// TwinCAT 3 PLC project VFD
// ProgramVersion: 3.1.4024.0
// libraries:
//   Modbus RTU Base, * (NewEngineer)
//   Tc2_ModbusRTU, * (Beckhoff Automation GmbH)
//   Tc2_Standard, * (Beckhoff Automation GmbH)
//   Tc2_System, * (Beckhoff Automation GmbH)
//   Tc3_Module, * (Beckhoff Automation GmbH)
//   TC3_Utilities_C, * (NewEngineer)
// project tree:
//   DUTs/ServoIpro/ E_IProCtrlMode.TcDUT (not stored), E_IProCurrentMode.TcDUT, E_IProStatus.TcDUT, E_IPro_PositionCmdModeSelection.TcDUT (not stored), E_IPro_State.TcDUT
//   DUTs/VFD/ E_VfdMdriverFaultInfor.TcDUT (not stored), E_VFD_State.TcDUT (not stored), E_VFD_Status.TcDUT (not stored)
//   / PlcTask.TcTTO
//   POUs/ FB_IPRO_ModbusRTU.TcPOU, FB_UniversalVFDModbus.TcPOU, FB_VFD_ABB_ACS480.TcPOU, FB_VFD_Mdriver.TcPOU, FB_VFD_V20_Siemens.TcPOU, I_Ipro_MotorPower.TcIO, I_UniversalVFD.TcIO, MAIN.TcPOU
//   TEST/ FB_ModbusMaster_Test.TcPOU (not stored), FB_ModbusSlave_Test.TcPOU (not stored), FB_UniversalVFDModbus_Ex.TcPOU (not stored), FB_UniversalVFDModbus_Test.TcPOU (not stored), PGR_Test.TcPOU (not stored)
// real-time tasks:
//   TASK PlcTask: cycle T#10ms, priority 20, ADS port 350

CONFIGURATION VFD
    RESOURCE PLC ON TwinCAT3
        TASK PlcTask(INTERVAL := T#10ms, PRIORITY := 20);
        PROGRAM MAIN WITH PlcTask : MAIN;
    END_RESOURCE
END_CONFIGURATION

// ---- DUTs/ServoIpro/E_IProCurrentMode.TcDUT
//{attribute 'strict'}
TYPE E_IProCurrentMode :
(
	IPRO_CURRENT_MODE_NOT_RESPONDE := -10,
	IPRO_CURRENT_MODE_POSITION		:= 0,
	IPRO_CURRENT_MODE_SPEED			:= 1,
	IPRO_CURRENT_MODE_TORQUE		:= 2
)INT := IPRO_CURRENT_MODE_NOT_RESPONDE;
END_TYPE

// ---- DUTs/ServoIpro/E_IProStatus.TcDUT
//{attribute 'strict'}
{attribute 'to_string'}
TYPE E_IProStatus :
(
	IPRO_STATUS_NOT_RESPOND := -10,
	IPRO_STATUS_INTITIZATION := 0,
	IPRO_STATUS_THE_HIGH_VOLTAGE := 1,
	IPRO_STATUS_READY			:= 2,
	IPRO_STATUS_RUN				:= 3, // OPERATION
	IPRO_STATUS_FORCED_TO_STOP	:= 4,
	IPRO_STATUS_FAULT			:= 5,
	IPRO_STATUS_STO_IN			:= 6
)INT := IPRO_STATUS_NOT_RESPOND;
END_TYPE

// ---- DUTs/ServoIpro/E_IPro_State.TcDUT
{attribute 'strict'}
{attribute 'to_string'}
TYPE E_IPro_State :
(
	IPRO_UNINITIALIZED		:= 0,	(* Axis is not prepared to work - power is off *)
	IPRO_INITIALIZING		:= 10,	(* Axis is preparing to power - reset FB and power on *)
	IPRO_READY_INITIALIZED		:= 20,	(*  *)
	IPRO_IDLE				:= 25,// MOVE DONE TO HERE
	IPRO_HOME			:= 30,	(* Axis is homing to reference point *)
	IPRO_HOME_DONE			:= 40,	(* Axis homing procedure has finished - fererence position has been found *)
	IPRO_MOVE_ABSOLUTE		:= 50,	(* Axis is moving to absolute position - discrete motion *)
	IPRO_MOVE_ABSOLUTE_DONE		:= 60,	(* Axis movement to absolute position finished *)
	IPRO_MOVE_TORQUE	:= 70,
	IPRO_MOVE_TORQUE_DONE	:= 80,
	//IPRO_MOVE_VELOCITY		:= 90,
	//IPRO_MOVE_VELOCITY_DONE	:= 100
	IPRO_STOP			:= 90,	(* Axis is stopping *)
	IPRO_STOP_DONE			:= 100,	(* Axis stopped *)
	IPRO_RESET			:= 110,	(* Axis is resseting all function blocks and occured errors *)
	IPRO_RESET_DONE			:= 120,	(* Axis reset procedure done *)
	IPRO_ABORTING			:= -10	(* Aborting *)
);
END_TYPE

// ---- POUs/I_Ipro_MotorPower.TcIO
INTERFACE I_Ipro_MotorPower

PROPERTY Active : bool
GET
END_GET
END_PROPERTY

PROPERTY Busy : bool
GET
END_GET
END_PROPERTY

PROPERTY ControlMode : E_IProCtrlMode
GET
END_GET
SET
END_SET
END_PROPERTY

PROPERTY ControlModeSwitchCmd : bool
GET
END_GET
END_PROPERTY

PROPERTY CurrentMode : E_IProCurrentMode
GET
END_GET
END_PROPERTY

PROPERTY Enable : bool
GET
END_GET
END_PROPERTY

PROPERTY Error : bool
GET
END_GET
END_PROPERTY

PROPERTY ErrorID : REFERENCE TO INT
GET
END_GET
END_PROPERTY

PROPERTY InPosition : bool
GET
END_GET
END_PROPERTY

PROPERTY IsInTorque : bool
GET
END_GET
END_PROPERTY

PROPERTY isStop : bool
GET
END_GET
END_PROPERTY

PROPERTY MaxSpeed : lreal// large than 0
GET
END_GET
SET
END_SET
END_PROPERTY

PROPERTY MaxTorque : Lreal// // % larger than 0
GET
END_GET
SET
END_SET
END_PROPERTY

METHOD MR_Abort : BOOL
END_METHOD

METHOD MR_Home : BOOL // control mode must have Position Mode // actually it the same as MOVE absolute 
VAR_INPUT
	lrHomePosition : LREAL;
END_VAR
END_METHOD

(*this must be called 2 times, first: after set All parram in "SetBefor Init" folder and before run FBModbusMaster
							 second : after Modbusmster running and state machine in Init state.*)
METHOD MR_Init : BOOL// need to set control mode carefully, the control mode only work correct if you set p0.03 and restart the driver, and there for if you change control mode cmd during driver power ON, the control mode will not effect
END_METHOD

METHOD MR_MoveAbsolute : BOOL // control mode must have Position Mode
VAR_INPUT
	lrAbsolutePosition : LREAL;
END_VAR
END_METHOD

METHOD MR_MoveTorque : BOOL // control mode must have torque Mode
VAR_INPUT
	lrTorque	: LREAL;// must smaller than max torque
END_VAR
END_METHOD

METHOD MR_Reset : BOOL// can't not use this method because i didn't find way to reset
END_METHOD

METHOD MR_Stop : BOOL
END_METHOD

PROPERTY NagativePositionLimit : lreal
GET
END_GET
SET
END_SET
END_PROPERTY

PROPERTY PositionCmd : lreal
GET
END_GET
END_PROPERTY

PROPERTY PositionFeedBack : lreal
GET
END_GET
END_PROPERTY

PROPERTY PositionModeSelectionCmd : E_IPro_PositionCmdModeSelection
GET
END_GET
END_PROPERTY

PROPERTY PositionModeSelectionFeedback : E_IPro_PositionCmdModeSelection
GET
END_GET
END_PROPERTY

PROPERTY PositionPositiveLimit : lreal
GET
END_GET
SET
END_SET
END_PROPERTY

PROPERTY SpeedCmd : LREAL // r/ minute
GET
END_GET
SET
END_SET
END_PROPERTY

PROPERTY SpeedFeedback : Lreal
GET
END_GET
END_PROPERTY

PROPERTY State : E_IPro_State
GET
END_GET
END_PROPERTY

PROPERTY Status : E_IProStatus
GET
END_GET
END_PROPERTY

PROPERTY TorqueCmd : lreal // %
GET
END_GET
END_PROPERTY

PROPERTY TorqueFeedback : lreal
GET
END_GET
END_PROPERTY

END_INTERFACE

// ---- POUs/I_UniversalVFD.TcIO
INTERFACE I_UniversalVFD


PROPERTY Active : REFERENCE TO  bool
GET
END_GET
END_PROPERTY

PROPERTY AcVoltageToMotor : Reference to lreal
GET
END_GET
END_PROPERTY


PROPERTY Busy : reference to bool
GET
END_GET
END_PROPERTY

PROPERTY Current : reference to lreal
GET
END_GET
END_PROPERTY

PROPERTY DcVoltage : Reference to lreal
GET
END_GET
END_PROPERTY


PROPERTY Error : REFERENCE to bool
GET
END_GET
END_PROPERTY


PROPERTY ErrorID : reference to UDINT
GET
END_GET
END_PROPERTY

PROPERTY HzActual : REFERENCE TO  LReal
GET
END_GET
END_PROPERTY

PROPERTY HzControl : reference to LReal
GET
END_GET
END_PROPERTY


PROPERTY InHz : bool
GET
END_GET
END_PROPERTY

PROPERTY isRunForward : bool
GET
END_GET
END_PROPERTY


PROPERTY IsRunning : bool
GET
END_GET
END_PROPERTY

PROPERTY isRunReverse : bool
GET
END_GET
END_PROPERTY

PROPERTY isStop : bool
GET
END_GET
END_PROPERTY

METHOD MR_Abort : BOOL
VAR_INPUT
END_VAR
END_METHOD

METHOD MR_Init : bool
VAR_INPUT
END_VAR
END_METHOD

METHOD MR_Reset : BOOL
VAR_INPUT
END_VAR
END_METHOD

//must stop before call run reverse or forward
METHOD MR_RunForward : BOOL// carefully about this state , it only into run forward if estatus = VFD_STATUS_RUNNING_FORWARD or it return True
VAR_INPUT
	hz : LREAL;
END_VAR
END_METHOD

METHOD MR_RunReverse : BOOL// must stop before call run reverse or forward
VAR_INPUT
	hz : LREAL; // >0 and < 50;
END_VAR
END_METHOD

METHOD MR_Stop : BOOL
VAR_INPUT
END_VAR
END_METHOD

PROPERTY Name : STRING
GET
END_GET
SET
END_SET
END_PROPERTY


PROPERTY Overload : reference TO BOOL
GET
END_GET
END_PROPERTY


PROPERTY PowerKw : REFERENCE TO LREAL
GET
END_GET
END_PROPERTY

PROPERTY ReallyError : bool
GET
END_GET
END_PROPERTY

PROPERTY Speed : Reference to lreal
GET
END_GET
END_PROPERTY


PROPERTY State : reference to E_Vfd_State
GET
END_GET
END_PROPERTY


PROPERTY Status : reference to E_VFD_Status
GET
END_GET
END_PROPERTY

PROPERTY timeStopDelay : time
GET
END_GET
SET
END_SET
END_PROPERTY

PROPERTY Torque : reference to lreal
GET
END_GET
END_PROPERTY

PROPERTY TotalKwh : reference to lreal
GET
END_GET
END_PROPERTY

PROPERTY Warning : reference to bool
GET
END_GET
END_PROPERTY

END_INTERFACE

// ---- POUs/MAIN.TcPOU
PROGRAM MAIN
VAR
	fbModbusMaster : MODBUSRTU.FB_ModbusMaster_PcCOM;
	fbabb : FB_VFD_ABB_ACS480;
	fbmdrive : FB_VFD_Mdriver;
	fbSiemen	: FB_VFD_V20_Siemens;
	fb_ipro	: FB_IPRO_ModbusRTU;
	
END_VAR

END_PROGRAM

// ---- POUs/FB_VFD_ABB_ACS480.TcPOU
FUNCTION_BLOCK FB_VFD_ABB_ACS480 EXTENDS FB_UniversalVFDModbus

VAR
	VFD_CTRL_RUN_EMERGENCY_STOP : WORD;
	TempData0: U_Word2Int;
END_VAR

SUPER^();

METHOD Convert : BOOL
VAR_INPUT
	iRegionNo	:	INT;
	pReadData	:	POINTER TO word;
END_VAR
CASE	iRegionNo OF

	0: // status
		IF pReadData[0].15 = TRUE THEN
			eVfdStatus := VFD_STATUS_FAULT;
			
		ELSIF (eVfdState = VFD_INITIALIZING
			OR eVfdState = VFD_READY_INITIALIZED)
			AND pReadData[0].0 = TRUE
			AND pReadData[0].1 = TRUE	
			AND pReadData[0].2 = TRUE
			THEN
			eVfdStatus :=  VFD_STATUS_READY_TO_RUN;
				
		ELSIF pReadData[0].3 = FALSE THEN
			eVfdStatus :=  VFD_STATUS_STOP;
			
		ELSIF pReadData[0].3 = TRUE	//run
			AND pReadData[0].10 = FALSE	// Drive reference is in the forward direction	
			AND pReadData[0].11 = FALSE//Drive is running in the forward direction
			THEN		
			eVfdStatus := VFD_STATUS_RUNNING_FORWARD;
		
		ELSIF pReadData[0].3 = TRUE	//run
			AND pReadData[0].10 = TRUE	// Drive reference is in the forward direction	
			AND pReadData[0].11 = TRUE//Drive is running in the forward direction
			THEN		
			eVfdStatus := VFD_STATUS_RUNNING_REVERSE;
		
		END_IF
	1: 
		TempData0.iWord := pReadData[0];
		lrHzActual		:= ABS(INT_TO_LREAL( TempData0.iInt)*0.0025);//50/20000;	
		lrCurrent		:= WORD_TO_LREAL( pReadData[1])*0.01;	//46.05 = 100
		lrDcVoltage		:= WORD_TO_LREAL( pReadData[5])*0.1;	
	
	2: 
		lrVacOutToMotor	:= WORD_TO_LREAL( pReadData[0]);	//4099	/1
		lrPowerKw		:= WORD_TO_LREAL( pReadData[1])*0.01;		//46.04
	
	3:
		lrTotalKwh :=  WORD_TO_LREAL( pReadData[0])*0.1;
		
	4: 
		lrSpeed :=  WORD_TO_LREAL( pReadData[0]);
	
	


END_CASE
END_METHOD

METHOD  FirstCycle 
VAR_INPUT
	sName : STRING;
	iUnitID : BYTE ; // modbus address of the device : 1- 255
END_VAR
SUPER^.FirstCycle( sName := sName, iUnitID := iUnitID);
(*Assign Ctrol Word : user Manual M-driver*)
VFD_CTRL_RESET_FAULT := 2#0001_0001;
VFD_CTRL_RUN_FORWARD := 2#0000_0010;
VFD_CTRL_RUN_REVERSE := 2#0000_0110;
VFD_CTRL_STOP_FREE 	 := 2#0010_0000_0001;
VFD_CTRL_STOP_SPEED_DOWN := 2#1000_0001;
VFD_CTRL_RUN_EMERGENCY_STOP := 2#0001_0000_0001;

// actual state	
	arrAddressRead[0][0] := 3;
	arrAddressRead[0][1] := 1;
	arrAddressRead[0][2] := E_ModbusFunction.ReadHoldingRegisters;

//mode0 address = 40000 + function*100 + sub function -1
	// actual hz  
	arrAddressRead[1][0] := 105; // 01.06
	arrAddressRead[1][1] := 6;
	arrAddressRead[1][2] := E_ModbusFunction.ReadHoldingRegisters;
	
	arrAddressRead[2][0] := 112; // 01.13
	arrAddressRead[2][1] := 2;
	arrAddressRead[2][2] := E_ModbusFunction.ReadHoldingRegisters;
	
	arrAddressRead[3][0] := 119; // 01.20
	arrAddressRead[3][1] := 1;
	arrAddressRead[3][2] := E_ModbusFunction.ReadHoldingRegisters;
	
	arrAddressRead[4][0] := 101; // 01.20
	arrAddressRead[4][1] := 1;
	arrAddressRead[4][2] := E_ModbusFunction.ReadHoldingRegisters;
iNumAddRegionRead	:= 5;

/////write control WORD VFD, // use ctrol word and frequency in 1 modbus write
arrAddressWrite[iCTRL_WORD][0]	:= 0;
arrAddressWrite[iCTRL_WORD][1]	:= 2;
arrAddressWrite[iCTRL_WORD][2]	:= VFD_CTRL_STOP_FREE;
arrAddressWrite[iCTRL_WORD][10]	:= E_ModbusFunction.WriteMultipleRegisters;

// Frequency
//arrAddressWrite[iCTRL_FREQUENCY_WORD][0]	:= 1;
//arrAddressWrite[iCTRL_FREQUENCY_WORD][1]	:= 1;
							(*MUST BE CARE FULL WHEN USE FLOATING POINT CONVERT*)
arrAddressWrite[iCTRL_FREQUENCY_WORD][3]	:= LREAL_TO_WORD( FC_ScaleValue(	rangeRawMin := 0,
																				rangeRawMax := 50,
																				RangeScaleMin :=0,
																				RangeScaleMax := 20000,
																				ValueRaw := 0)
										  );
										  
iNumAddRegionWrite := 1;// use ctrol word and frequency in 1 modbus write
END_METHOD

METHOD PROTECTED  MS_Aborting
arrAddressWrite[iCTRL_WORD][2]	:= VFD_CTRL_STOP_FREE;
SUPER^.MS_Aborting();
END_METHOD

METHOD  PROTECTED  MS_Initializing
SUPER^.MS_Initializing();
END_METHOD

METHOD PROTECTED  MS_RunForward
VAR_INPUT
END_VAR
// use ctrol word and frequency in 1 modbus write WRITE MULTIES REGIS
arrAddressWrite[iCTRL_WORD][3] :=  LREAL_TO_WORD( 
															FC_ScaleValue(	rangeRawMin := 0,
																			rangeRawMax := 50,
																			RangeScaleMin := 0,
																			RangeScaleMax := 20000,
																			ValueRaw := lrHzControl) 
																				);
SUPER^.MS_RunForward();
END_METHOD

METHOD PROTECTED  MS_RunReverse
VAR_INPUT
END_VAR
// use ctrol word and frequency in 1 modbus write WRITE MULTIES REGIS
arrAddressWrite[iCTRL_WORD][3] :=  LREAL_TO_WORD( 
															FC_ScaleValue(	rangeRawMin := 0,
																			rangeRawMax := 50,
																			RangeScaleMin := 0,
																			RangeScaleMax := 20000,
																			ValueRaw := lrHzControl) 
																				);
SUPER^.MS_RunReverse();
END_METHOD

END_FUNCTION_BLOCK

// ---- POUs/FB_UniversalVFDModbus.TcPOU
FUNCTION_BLOCK abstract FB_UniversalVFDModbus EXTENDS FB_ModbusSlave IMPLEMENTS I_UniversalVFD
VAR
	eVfdState	: E_Vfd_State;
	bInit	: BOOL;
	bBusy	: BOOL;
	bReset	: BOOL;
	bStop	: BOOL;
	bAbort : BOOL;
	bError : BOOL;
	bWarning : BOOL;// status
	bRunningForward	: BOOL;// in state running forward
	bRunningReverse	: BOOL; // in state running reverse
	bRanForward	: BOOL;
	bRanReverse	: BOOL;
	lrHzActual	: LREAL;
	lrDcVoltage		: LREAL;
	lrVacOutToMotor	: LREAL;
	lrCurrent	: LREAL;	
	lrPowerKw	: LREAL;	
	eVfdStatus	: E_VFD_Status;
	lrHzControl	: LREAL;// value in range(0.0-50.0Hz)
	iErrorID		: UDINT;

	lrSpeed : LREAL;
	lrTorque : LREAL;
	lrTotalKwh : LREAL;
	lrRatedPower : LREAL;
	bActive: BOOL;
	bOverLoad: BOOL;
	bStopLog: BOOL;
	bStopped: BOOL;
	
	VFD_CTRL_RESET_FAULT : WORD;
	VFD_CTRL_RUN_FORWARD :WORD;
	VFD_CTRL_RUN_REVERSE :WORD ;
	VFD_CTRL_STOP_FREE 		:WORD ;
	VFD_CTRL_STOP_SPEED_DOWN	:WORD ;
	
	tonStopDelay: Ton;
	// time delay after status = stop
	tStopDelay: TIME := T#4S;
	bReallyError	: BOOL;// because of bError maybe incorrect because noise information return by Modbus
	tonConfirmReallyError : TON;
	timeConfirmReallyError : TIME := T#15S;
END_VAR
VAR CONSTANT
	// index
	iCTRL_WORD	: UINT := 1;
	iCTRL_FREQUENCY_WORD :UINT := 0;
	iSTATUS_WORD	: UINT := 0;
END_VAR

StateMachine();
CASE eVfdStatus OF
	VFD_STATUS_RUNNING_FORWARD :
		bRanForward := TRUE;
		bRanReverse := FALSE;
		bStopped := FALSE;
	VFD_STATUS_RUNNING_REVERSE:
		bRanForward := FALSE;
		bRanReverse := TRUE;
		bStopped := FALSE;
	VFD_STATUS_FAULT,VFD_STATUS_STOP:
		bRanForward := FALSE;
		bRanReverse := FALSE;
		bStopped := TRUE;
		
END_CASE
bError := eVfdStatus = VFD_STATUS_FAULT;
bActive := eVfdState >= VFD_IDLE;
CASE eVfdState OF
	VFD_INITIALIZING..VFD_RESET_DONE, VFD_ABORTING:
		tonConfirmReallyError(
			IN := bError OR iModbusErrorID <> MODBUSERROR_NO_ERROR,
			PT := timeConfirmReallyError,
			Q => bReallyError 
		);
END_CASE

{attribute 'monitoring' := 'variable'}
PROPERTY Active : REFERENCE TO  bool
GET
Active REF= bActive;
END_GET
END_PROPERTY

PROPERTY AcVoltageToMotor : Reference to lreal
GET
AcVoltageToMotor ref= lrVacOutToMotor;
END_GET
END_PROPERTY

{attribute 'monitoring' := 'variable'}
PROPERTY Busy : reference to bool
GET
Busy ref= bBusy;
END_GET
END_PROPERTY

METHOD Convert : BOOL
VAR_INPUT
	iRegionNo	:	INT;
	pReadData	:	POINTER TO word;
END_VAR
(*CASE iRegionNo OF
	0:
		// Status word
		Inverter_Ready		:=  pReadData[0].0;
		InverterReadyToRun	:=  pReadData[0].1;
		InverterRunning		:=  pReadData[0].2;
		InverterFaultActive :=  pReadData[0].3;
		OFF2_active			:= NOT pReadData[0].4;
		OFF3_active			:= NOT  pReadData[0].5;
		ON_inhibit_active 	 := pReadData[0].6;
		Inverter_warning_active := pReadData[0].7;
		Deviation_setpoint_OR_ActiveValue := NOT pReadData[0].8;
		PZD_control 		:= pReadData[0].9;
		Motor_current_Or_torque_limit  := NOT pReadData[0].11;
		Brake_open	 := pReadData[0].12;
		Motor_overload := NOT pReadData[0].13;
		Motor_RunRight	:= pReadData[0].14;
		Inverter_overload :=  NOT pReadData[0].15;
		
		IF InverterFaultActive THEN
			eStatus := VFD_STATUS_FAULT;
		ELSIF InverterFaultActive THEN
			eStatus := VFD_STATUS_WARNING;
		ELSIF InverterRunning THEN
			IF Motor_RunRight THEN
				eStatus := VFD_STATUS_RUNNING_FORWARD;
			ELSE
				eStatus := VFD_STATUS_RUNNING_REVERSE;
			END_IF
		ELSIF NOT InverterRunning THEN
			eStatus := VFD_STATUS_STOP;
		END_IF

		// Speed word
		lrHz_actual := WORD_TO_LREAL( pReadData[1])*50/16383;
		
	1:
		///  actual  Speed ( rpm) (unit A : Scale factor 1), Current ( A , 100, , Torque (Nm, 100)
	//, Actual Power (kw, 100), Total Kwh( 1), Dc bus Voltage(1), REFERENCE( hz, 100), RATED PWR( 100),OUTPUT VOLTS(1)
		lrSpeed := pReadData[0];
		lrCurrent := WORD_TO_LREAL(pReadData[1])/100;
		lrTorque := WORD_TO_LREAL(pReadData[2])/100;
		lrPower := WORD_TO_LREAL(pReadData[3])/100;
		lrTotalKwh := WORD_TO_LREAL(pReadData[4]);
		lrDc_Voltage := WORD_TO_LREAL(pReadData[5]);
		lrRatedPower := WORD_TO_LREAL(pReadData[7])/100;
		lrVAC_OutToMotor := WORD_TO_LREAL(pReadData[8]);
END_CASE
*)
END_METHOD

PROPERTY Current : reference to lreal
GET
Current ref= lrCurrent;
END_GET
END_PROPERTY

PROPERTY DcVoltage : Reference to lreal
GET
DcVoltage ref= lrDcVoltage;
END_GET
END_PROPERTY

{attribute 'monitoring' := 'variable'}
PROPERTY Error : REFERENCE to bool
GET
Error ref= bError;
END_GET
END_PROPERTY

{attribute 'monitoring' := 'variable'}
PROPERTY ErrorID : reference to UDINT
GET
ErrorID ref= iErrorID;
END_GET
END_PROPERTY

METHOD  FirstCycle 
VAR_INPUT
	sName : STRING;
	iUnitID : BYTE ; // modbus address of the device : 1- 255
END_VAR
THIS^.sName := sName;
THIS^.iUnitID := iUnitID;
(*(*HSW (speed setpoint), HIW (actual speed), STW (control word), ZSW (status word) refer to
control data. For more information, see parameters r2018 and P2019 in Chapter "Parameter
list (Page 147)*)
//ZSW  (status WORD), HIW (actual speed)
	arrAddress[0][0] := 109;
	arrAddress[0][1]	:= 2;

///  actual  Speed ( rpm) (unit A : Scale factor 1), Current ( A , 100, , Torque (Nm, 100)
	//, Actual Power (kw, 100), Total Kwh( 1), Dc bus Voltage(1), REFERENCE( hz, 100), RATED PWR( 100),OUTPUT VOLTS(1)
	arrAddress[1][0] := 24;
	arrAddress[1][1] := 10;

	
iNumAddRegion	:= 2;
/////write control  VFD
	
// Frequency

arrAddressWrite[0][0]	:= 100;
arrAddressWrite[0][1] 	:= 1;
arrAddressWrite[0][2]	:= LREAL_TO_WORD( FC_ScaleValue(	rangeRawMin := 0,
															rangeRawMax := 50,
															RangeScaleMin :=0,
															RangeScaleMax := 16384,
															ValueRaw := lrHz_Control) );
// Control word																	
arrAddressWrite[1][0]	:= 99;
arrAddressWrite[1][1] := 1;
arrAddressWrite[1][2]	:= 1150; //VFD_CTRL_STOP_SPEED_DOWN
iNumAddRegionWrite := 2;
*)
END_METHOD

PROPERTY HzActual : REFERENCE TO  LReal
GET
HzActual ref= lrHzActual;
END_GET
END_PROPERTY

PROPERTY HzControl : reference to LReal
GET
HzControl ref= lrHzControl;
END_GET
END_PROPERTY

{attribute 'monitoring' := 'variable'}
PROPERTY InHz : bool
GET
InHz :=  FC_InRange( bound1 := lrHzControl +1,
					bound2 := lrHzControl -1,
					value := lrHzActual) ;
END_GET
END_PROPERTY

PROPERTY isRunForward : bool
GET
isRunForward := bRanForward;
END_GET
END_PROPERTY

{attribute 'monitoring' := 'variable'}
PROPERTY IsRunning : bool
GET
IsRunning := eVfdStatus = VFD_STATUS_RUNNING_FORWARD
			 OR  eVfdStatus = VFD_STATUS_RUNNING_REVERSE;
END_GET
END_PROPERTY

PROPERTY isRunReverse : bool
GET
isRunReverse := bRanReverse;
END_GET
END_PROPERTY

PROPERTY isStop : bool
GET
isStop := bStopped;
END_GET
END_PROPERTY

METHOD MR_Abort : BOOL
VAR_INPUT
END_VAR
IF eVfdState >= VFD_INITIALIZING THEN
	bAbort := TRUE;
	eVfdState := VFD_ABORTING;
	fbMachineLogger.MR_AddLogs(CONCAT(sName,' : abort requested'));
	bBusy := TRUE;
	
ELSIF eVfdState = VFD_UNINITIALIZED THEN
	bAbort 		:= FALSE;
	MR_Abort	:= TRUE;
	bBusy := FALSE;
	fbMachineLogger.MR_AddLogs(CONCAT(sName,' : abort done'));
	
END_IF
END_METHOD

METHOD MR_Init : bool
VAR_INPUT
END_VAR
IF eVFDState = VFD_UNINITIALIZED THEN
	bInit := TRUE;
	MR_Init := FALSE;
	eVfdState := VFD_INITIALIZING;
	fbMachineLogger.MR_AddLogs(CONCAT(sName,' : initialization requested'));
	bBusy := TRUE;
	
ELSIF eVFDState = VFD_READY_INITIALIZED THEN
	bInit := FALSE;
	MR_Init := TRUE;
	bBusy := FALSE;
	fbMachineLogger.MR_AddLogs(CONCAT(sName,' : initialization done'));
END_IF
END_METHOD

METHOD MR_Reset : BOOL
VAR_INPUT
END_VAR
IF eVfdState >= VFD_IDLE AND bError THEN
	bReset := TRUE;
	eVfdState := VFD_RESET;
	fbMachineLogger.MR_AddLogs(CONCAT(sName,' : reset requested'));			
	bBusy := TRUE;
	
ELSIF eVfdState = VFD_RESET_DONE THEN
	bError := FALSE;
	iErrorID := 0;
	bReset := FALSE;
	MR_Reset := TRUE;
	bBusy := FALSE;
	fbMachineLogger.MR_AddLogs(CONCAT(sName,' : reset done'));		
		
END_IF
END_METHOD

METHOD MR_RunForward : BOOL
VAR_INPUT
	hz : LREAL; 
END_VAR
IF eVfdState = VFD_IDLE  AND (NOT  FC_InRange( 	bound1 := lrHzControl + 0.01,
												bound2 := lrHzControl - 0.01,
												value :=  hz)
								OR bRanReverse
								OR bStopped)
THEN
	lrHzControl := hz;
	bRunningForward := TRUE;
	MR_RunForward := FALSE;
	eVfdState := VFD_RUN_FORWARD;
	fbMachineLogger.MR_AddLogs( sLogMessage := FUN_MergeStrings4(  sName,' : run ',LREAL_TO_STRING( lrHzControl),' forward requested'));		
	bBusy := TRUE;
	
ELSIF eVfdState = VFD_RUN_FORWARD_DONE THEN
	bRunningForward := FALSE;
	MR_RunForward := TRUE;
	fbMachineLogger.MR_AddLogs(CONCAT(sName,' : run forward done'));	
	bBusy := FALSE;
END_IF
END_METHOD

METHOD MR_RunReverse : BOOL// must stop before call run reverse or forward
VAR_INPUT
	hz : LREAL; // >0 and < 50;
END_VAR
IF eVfdState = VFD_IDLE  AND (NOT  FC_InRange( 	bound1 := lrHzControl + 0.01,
												bound2 := lrHzControl - 0.01,
												value :=  hz)
								OR bRanForward
								OR bStopped)
THEN
	lrHzControl := hz;
	bRunningReverse := TRUE;
	MR_RunReverse := FALSE;
	eVfdState := VFD_RUN_REVERSE;
	fbMachineLogger.MR_AddLogs( sLogMessage := FUN_MergeStrings4(  sName,' : run ',LREAL_TO_STRING( lrHzControl),' forward requested'));		
	bBusy := TRUE;
	
ELSIF eVfdState = VFD_RUN_REVERSE_DONE THEN
	bRunningReverse := FALSE;
	MR_RunReverse := TRUE;
	fbMachineLogger.MR_AddLogs(CONCAT(sName,' : run forward done'));
	bBusy := FALSE;
END_IF
END_METHOD

METHOD MR_Stop : BOOL
VAR_INPUT
END_VAR
IF eVfdState >= VFD_IDLE AND eVfdState <> VFD_STOP_DONE THEN
	IF NOT bStopLog THEN 
		fbMachineLogger.MR_AddLogs(CONCAT(sName,' : stop requested'));
		bStopLog := TRUE;	
	END_IF
	
	bStop := TRUE;
	eVfdState := VFD_STOP;
	bBusy := TRUE;
	
ELSIF eVfdState = VFD_STOP_DONE THEN
	bStop 		:= FALSE;
	MR_Stop 	:= TRUE;
	bStopLog 	:= FALSE;
	fbMachineLogger.MR_AddLogs(CONCAT(sName,' : stop done'));	
	bBusy := FALSE;
END_IF
END_METHOD

METHOD PROTECTED MS_Aborting
lrHzControl := 0;
bInit := FALSE;
bRunningForward := FALSE;
bRunningReverse := FALSE;
bReset := FALSE;
bRanForward := FALSE;
bRanReverse := FALSE;
bOverLoad := FALSE;
bStop := FALSE;
bStopLog := FALSE;
bStopped := FALSE;
THIS^.tonStopDelay(IN :=FALSE);
IF eVfdStatus = VFD_STATUS_STOP OR eVfdStatus = VFD_STATUS_FAULT THEN
	eVfdState := VFD_UNINITIALIZED;
END_IF
END_METHOD

METHOD PROTECTED MS_Idle
;
END_METHOD

METHOD  PROTECTED  MS_Initializing
// from Subclass call Super^.MS_Initializing
arrAddressWrite[iCTRL_WORD][2]	:= VFD_CTRL_RESET_FAULT;
IF eVfdStatus = VFD_STATUS_READY_TO_RUN THEN
	eVFDState := VFD_READY_INITIALIZED;
END_IF
END_METHOD

METHOD PROTECTED MS_ReadyInitialized
VAR_INPUT
END_VAR
IF NOT bInit THEN
	eVfdState := VFD_IDLE;
END_IF
END_METHOD

METHOD PROTECTED  MS_Reset
VAR_INPUT
END_VAR
arrAddressWrite[iCTRL_WORD][2]	:= VFD_CTRL_RESET_FAULT;
IF THIS^.evfdStatus <>  VFD_STATUS_NOT_RESPOND AND
	THIS^.evfdStatus <>  VFD_STATUS_FAULT THEN
	evfdState := VFD_RESET_DONE;
END_IF
END_METHOD

METHOD PROTECTED MS_ResetDone
VAR_INPUT
END_VAR
IF NOT bReset THEN
	evfdState := VFD_IDLE;
END_IF
END_METHOD

METHOD PROTECTED  MS_RunForward
VAR_INPUT
END_VAR
(*arrAddressWrite[iCtrlFrequencyWord][2] :=  LREAL_TO_WORD( 
											FC_ScaleValue(		rangeRawMin := 0,
																rangeRawMax := 50,
																RangeScaleMin := WORD_TO_LREAL( wHzWordValueMin),
																RangeScaleMax := WORD_TO_LREAL( wHzWordValueMax),
																ValueRaw := lrHzControl) 
														);*)
arrAddressWrite[iCTRL_WORD][2]	:= VFD_CTRL_RUN_FORWARD;
IF eVfdStatus = VFD_STATUS_RUNNING_FORWARD 
(*AND F_InRange( bound1 := lrHzControl + 1,
				bound2 := lrHzControl -1,
				value := lrHzActual)*)
THEN
	eVFDState := VFD_RUN_FORWARD_DONE;
END_IF
END_METHOD

METHOD PROTECTED MS_RunForwardDone
IF NOT bRunningForward THEN
	eVfdState := VFD_IDLE;
END_IF
END_METHOD

METHOD PROTECTED  MS_RunReverse
VAR_INPUT
END_VAR
(*arrAddressWrite[iCtrlFrequencyWord][2] :=  LREAL_TO_WORD( 
											FC_ScaleValue(		rangeRawMin := 0,
																rangeRawMax := 50,
																RangeScaleMin := WORD_TO_LREAL( wHzWordValueMin),
																RangeScaleMax := WORD_TO_LREAL( wHzWordValueMax),
																ValueRaw := lrHzControl) 
														);*)
arrAddressWrite[iCTRL_WORD][2]	:= VFD_CTRL_RUN_REVERSE;
IF eVfdStatus = VFD_STATUS_RUNNING_REVERSE 
(*AND F_InRange( bound1 := lrHzControl + 1,
				bound2 := lrHzControl -1,
				value := lrHzActual)*)
THEN
	eVFDState := VFD_RUN_REVERSE_DONE;
END_IF
END_METHOD

METHOD PROTECTED MS_RunReverseDone
VAR_INPUT
END_VAR
IF NOT bRunningReverse THEN
	eVfdState := VFD_IDLE;
END_IF
END_METHOD

METHOD protected  MS_Stop 
VAR_INPUT
END_VAR
arrAddressWrite[iCTRL_WORD][2]	:= VFD_CTRL_STOP_SPEED_DOWN;
(*tonStopDelay( in := eVfdStatus = VFD_STATUS_STOP,
				PT := tStopDelay);*)
IF eVfdStatus = VFD_STATUS_STOP THEN
 eVfdState := VFD_STOP_DONE;	
END_IF
(*IF tonStopDelay.Q THEN
	tonStopDelay(IN := FALSE);
	
END_IF*)
END_METHOD

METHOD protected Ms_StopDone
VAR_INPUT
END_VAR
IF NOT bStop THEN
	eVfdState := VFD_IDLE;
END_IF
END_METHOD

METHOD PROTECTED MS_Uninitialized
END_METHOD

{attribute 'monitoring' := 'variable'}
PROPERTY Overload : reference TO BOOL
GET
Overload REF= bOverLoad;
END_GET
END_PROPERTY

{attribute 'monitoring' := 'variable'}
PROPERTY PowerKw : REFERENCE TO LREAL
GET
PowerKw ref= lrPowerKw;
END_GET
END_PROPERTY

PROPERTY ReallyError : bool
GET
ReallyError := bReallyError;
END_GET
END_PROPERTY

PROPERTY Speed : Reference to lreal
GET
Speed REF= lrSpeed;
END_GET
END_PROPERTY

{attribute 'monitoring' := 'variable'}
PROPERTY State : reference to E_Vfd_State
GET
State REF= eVfdState;
END_GET
END_PROPERTY

METHOD PROTECTED StateMachine
CASE eVfdState OF
	VFD_UNINITIALIZED :
		MS_Uninitialized();
		
	VFD_INITIALIZING	:
		MS_Initializing();
		
	VFD_READY_INITIALIZED :
		MS_ReadyInitialized();
		
	VFD_IDLE:
		MS_Idle();
	
	VFD_RUN_FORWARD	:
		MS_RunForward();
		
	VFD_RUN_FORWARD_DONE:
		MS_RunForwardDone();
	
	VFD_RUN_REVERSE	:
		MS_RunReverse();
	
	VFD_RUN_REVERSE_DONE:
		MS_RunReverseDone();
	
	VFD_STOP		:
		MS_Stop();
		
	VFD_STOP_DONE	:
		Ms_StopDone();
		
	VFD_RESET	:
		MS_Reset();
		
	VFD_RESET_DONE	:
		MS_ResetDone();
		
	VFD_ABORTING :
		MS_Aborting();
	
	
END_CASE
END_METHOD

{attribute 'monitoring' := 'variable'}
PROPERTY Status : reference to E_VFD_Status
GET
Status REF= eVfdStatus;
END_GET
END_PROPERTY

PROPERTY TimeRemainConfirmReallyError : Time
GET
TimeRemainConfirmReallyError := timeConfirmReallyError;
END_GET
SET
timeConfirmReallyError := TimeRemainConfirmReallyError;
END_SET
END_PROPERTY

PROPERTY timeStopDelay : time
GET
timeStopDelay := THIS^.tStopDelay;
END_GET
SET
tStopDelay := timeStopDelay;
END_SET
END_PROPERTY

PROPERTY Torque : reference to lreal
GET
Torque ref= Torque;
END_GET
END_PROPERTY

PROPERTY TotalKwh : reference to lreal
GET
TotalKwh REF= TotalKwh;
END_GET
END_PROPERTY

// not all vfd modbus available this function 
PROPERTY Warning : reference to bool
GET
Warning  ref= bWarning;
END_GET
END_PROPERTY

END_FUNCTION_BLOCK

// ---- POUs/FB_VFD_Mdriver.TcPOU
FUNCTION_BLOCK FB_VFD_Mdriver EXTENDS FB_UniversalVFDModbus

VAR
	eFaultInfor	: E_VfdMdriverFaultInfor;
END_VAR

//bError := eVfdStatus
SUPER^();

METHOD Convert : BOOL
VAR_INPUT
	iRegionNo	:	INT;
	pReadData	:	POINTER TO word;
END_VAR
CASE	iRegionNo OF
	0: 
	
		lrHzActual		:= WORD_TO_LREAL( pReadData[0])*0.01;	//4097	/unit /100
		lrDcVoltage		:= WORD_TO_LREAL( pReadData[1])*0.1;	//4098 	/10
		lrVacOutToMotor	:= WORD_TO_LREAL( pReadData[2]);	//4099	/1
		lrCurrent		:= WORD_TO_LREAL(  pReadData[3])*0.01;		//4100	/100
		//4 reserve
		lrPowerKw		:= WORD_TO_LREAL(  pReadData[5])*0.001;		//4102	/1000> kW
	
	1: // status
		CASE pReadData[0] OF
			0: eVfdStatus := VFD_STATUS_STOP;
			
			1: 
				eVfdStatus := VFD_STATUS_RUNNING_FORWARD;
			2:
				eVfdStatus := VFD_STATUS_RUNNING_REVERSE;
			3: 
				eVfdStatus := VFD_STATUS_STOP;
		END_CASE
		// important
		IF eVfdState = VFD_INITIALIZING THEN
			IF eFaultInfor = E_VfdMdriverFaultInfor.Nofault
			AND eVfdStatus = VFD_STATUS_STOP THEN
				eVfdStatus := VFD_STATUS_READY_TO_RUN;
			ELSIF eFaultInfor <> E_VfdMdriverFaultInfor.Nofault THEN
				eVfdStatus := VFD_STATUS_FAULT;
			END_IF
		END_IF
		IF eFaultInfor <> E_VfdMdriverFaultInfor.Nofault THEN
			eVfdStatus := VFD_STATUS_FAULT;
		END_IF
		IF iModbusErrorID = MODBUSERROR_NO_RESPONSE THEN
			eVfdStatus := VFD_STATUS_NOT_RESPOND;
		END_IF
		// important
	
	2: 
	
		iErrorID := WORD_TO_UDINT( pReadData[0]);
		eFaultInfor :=  WORD_TO_UINT( pReadData[0]);
END_CASE
END_METHOD

METHOD  FirstCycle 
VAR_INPUT
	sName : STRING;
	iUnitID : BYTE ; // modbus address of the device : 1- 255
END_VAR
SUPER^.FirstCycle( sName := sName, iUnitID := iUnitID);
(*Assign Ctrol Word : user Manual M-driver*)
VFD_CTRL_RESET_FAULT := 7;
VFD_CTRL_RUN_FORWARD := 1;
VFD_CTRL_RUN_REVERSE := 2;
VFD_CTRL_STOP_FREE 		:= 5;
VFD_CTRL_STOP_SPEED_DOWN	:= 6;
///  actual hz, current, voltage
arrAddressRead[0][0] := 4097;
arrAddressRead[0][1]	:= 6;
arrAddressRead[0][2]	:= E_ModbusFunction.ReadHoldingRegisters;

// actual state	
arrAddressRead[1][0] := 16#3000;
arrAddressRead[1][1]	:= 1;
arrAddressRead[1][2]	:= E_ModbusFunction.ReadHoldingRegisters;

// fault infor
arrAddressRead[2][0] := 16#8000;
arrAddressRead[2][1]	:= 1;
arrAddressRead[2][2]	:= E_ModbusFunction.ReadHoldingRegisters;

iNumAddRegionRead	:= 3;

/////write control WORD VFD
arrAddressWrite[iCTRL_WORD][0]	:= 16#2000;
arrAddressWrite[iCTRL_WORD][1]	:= 1;
arrAddressWrite[iCTRL_WORD][2]	:= VFD_CTRL_STOP_FREE;
arrAddressWrite[iCTRL_WORD][10]	:= E_ModbusFunction.WriteSingleRegister;
// Frequency
arrAddressWrite[iCTRL_FREQUENCY_WORD][0]	:= 4096;
arrAddressWrite[iCTRL_FREQUENCY_WORD][1]	:= 1;
							(*MUST BE CARE FULL WHEN USE FLOATING POINT CONVERT*)
arrAddressWrite[iCTRL_FREQUENCY_WORD][2]	:= LREAL_TO_WORD( FC_ScaleValue(	rangeRawMin := 0,
															rangeRawMax := 50,
															RangeScaleMin :=0,
															RangeScaleMax := 10000,
															ValueRaw := 0)
										  );
arrAddressWrite[iCTRL_FREQUENCY_WORD][10]	:= E_ModbusFunction.WriteSingleRegister;
										  
iNumAddRegionWrite := 2;
END_METHOD

METHOD PROTECTED  MS_Aborting
arrAddressWrite[iCTRL_WORD][2]	:= VFD_CTRL_STOP_FREE;
SUPER^.MS_Aborting();
END_METHOD

METHOD PROTECTED  MS_RunForward
VAR_INPUT
END_VAR
arrAddressWrite[iCTRL_FREQUENCY_WORD][2] :=  LREAL_TO_WORD( 
															FC_ScaleValue(	rangeRawMin := 0,
																			rangeRawMax := 50,
																			RangeScaleMin := 0,
																			RangeScaleMax := 10000,
																			ValueRaw := lrHzControl) 
																				);
SUPER^.MS_RunForward();
END_METHOD

METHOD PROTECTED  MS_RunReverse
VAR_INPUT
END_VAR
arrAddressWrite[iCTRL_FREQUENCY_WORD][2] :=  LREAL_TO_WORD( 
															FC_ScaleValue(	rangeRawMin := 0,
																			rangeRawMax := 50,
																			RangeScaleMin := 0,
																			RangeScaleMax := 10000,
																			ValueRaw := lrHzControl) 
																				);
SUPER^.MS_RunReverse();
END_METHOD

END_FUNCTION_BLOCK

// ---- POUs/FB_VFD_V20_Siemens.TcPOU
FUNCTION_BLOCK FB_VFD_V20_Siemens EXTENDS FB_UniversalVFDModbus
VAR			
	// status word
	Inverter_Ready		: BOOL;
	InverterReadyToRun	: BOOL;
	InverterRunning		: BOOL;
	InverterFaultActive : BOOL;
	OFF2_active			: BOOL;
	OFF3_active			: BOOL;
	ON_inhibit_active 	 : BOOL;
	Inverter_warning_active : BOOL;
	Deviation_setpoint_OR_ActiveValue : BOOL;
	PZD_control 		: BOOL;
	Motor_current_Or_torque_limit  : BOOL;
	Brake_open	 : BOOL;
	Motor_overload : BOOL;
	Motor_RunRight	: BOOL;
	Inverter_overload :BOOL; 
	//mode
	///  actual  Speed ( rpm) (unit A : Scale factor 1), Current ( A , 100, , Torque (Nm, 100)
	//, Actual Power (kw, 100), Total Kwh( 1), Dc bus Voltage(1), REFERENCE( hz, 100), RATED PWR( 100),OUTPUT VOLTS(1)
END_VAR

SUPER^();

METHOD Convert : BOOL
VAR_INPUT
	iRegionNo	:	INT;
	pReadData	:	POINTER TO word;
END_VAR
CASE iRegionNo OF
	0:
		// Status word
		Inverter_Ready		:=  pReadData[0].0;
		InverterReadyToRun	:=  pReadData[0].1;
		InverterRunning		:=  pReadData[0].2;
		InverterFaultActive :=  pReadData[0].3;
		OFF2_active			:= NOT pReadData[0].4;
		OFF3_active			:= NOT  pReadData[0].5;
		ON_inhibit_active 	 := pReadData[0].6;
		Inverter_warning_active := pReadData[0].7;
		Deviation_setpoint_OR_ActiveValue := NOT pReadData[0].8;
		PZD_control 		:= pReadData[0].9;
		Motor_current_Or_torque_limit  := NOT pReadData[0].11;
		Brake_open	 := pReadData[0].12;
		Motor_overload := NOT pReadData[0].13;
		Motor_RunRight	:= pReadData[0].14;
		Inverter_overload :=  NOT pReadData[0].15;
		
		IF eVfdState = VFD_INITIALIZING AND Inverter_Ready THEN
			eVfdStatus := VFD_STATUS_READY_TO_RUN;
		ELSIF InverterFaultActive THEN
			eVfdStatus := VFD_STATUS_FAULT;
//		ELSIF InverterFaultActive THEN
//			eVfdStatus := VFD_STATUS_WARNING;
		ELSIF InverterRunning THEN
			IF Motor_RunRight THEN
				eVfdStatus := VFD_STATUS_RUNNING_FORWARD;
			ELSE
				eVfdStatus := VFD_STATUS_RUNNING_REVERSE;
			END_IF
		ELSIF NOT InverterRunning THEN
			eVfdStatus := VFD_STATUS_STOP;
		END_IF

		// Speed word
		lrHzactual := WORD_TO_LREAL( pReadData[1])*50/16383;
		
	1:
		///  actual  Speed ( rpm) (unit A : Scale factor 1), Current ( A , 100, , Torque (Nm, 100)
	//, Actual Power (kw, 100), Total Kwh( 1), Dc bus Voltage(1), REFERENCE( hz, 100), RATED PWR( 100),OUTPUT VOLTS(1)
		lrSpeed := pReadData[0];
		lrCurrent := WORD_TO_LREAL(pReadData[1])/100;
		lrTorque := WORD_TO_LREAL(pReadData[2])/100;
		lrPowerKw := WORD_TO_LREAL(pReadData[3])/100;
		lrTotalKwh := WORD_TO_LREAL(pReadData[4]);
		lrDcVoltage := WORD_TO_LREAL(pReadData[5]);
		lrRatedPower := WORD_TO_LREAL(pReadData[7])/100;
		lrVACOutToMotor := WORD_TO_LREAL(pReadData[8]);
END_CASE
END_METHOD

METHOD  FirstCycle 
VAR_INPUT
	sName : STRING;
	iUnitID : BYTE ; // modbus address of the device : 1- 255
END_VAR
THIS^.sName := sName;
THIS^.iUnitID := iUnitID;
VFD_CTRL_STOP_FREE		:= 2#010001111010; // casue fault , reset error to run again	
VFD_CTRL_RUN_FORWARD	:= 2#010001111111;	
VFD_CTRL_RUN_REVERSE	 := 2#110001111111;	
VFD_CTRL_STOP_SPEED_DOWN := 2#010001111110;
VFD_CTRL_RESET_FAULT	 := 2#010011111110;
(*HSW (speed setpoint), HIW (actual speed), STW (control word), ZSW (status word) refer to
control data. For more information, see parameters r2018 and P2019 in Chapter "Parameter
list (Page 147)*)

//ZSW  (status WORD), HIW (actual speed)
	arrAddressRead[0][0] := 109;
	arrAddressRead[0][1] := 2;
	arrAddressRead[0][2] := E_ModbusFunction.ReadHoldingRegisters;
///  actual  Speed ( rpm) (unit A : Scale factor 1), Current ( A , 100, , Torque (Nm, 100)
	//, Actual Power (kw, 100), Total Kwh( 1), Dc bus Voltage(1), REFERENCE( hz, 100), RATED PWR( 100),OUTPUT VOLTS(1)
	arrAddressRead[1][0] := 24;
	arrAddressRead[1][1] := 10;
	arrAddressRead[1][2] := E_ModbusFunction.ReadHoldingRegisters;
	
iNumAddRegionRead	:= 2;
/////write control  VFD
// Control word																	
arrAddressWrite[iCTRL_WORD][0]	:= 99;
arrAddressWrite[iCTRL_WORD][1]  := 1;
arrAddressWrite[iCTRL_WORD][2]	:= 1150; //VFD_CTRL_STOP_SPEED_DOWN
arrAddressWrite[iCTRL_WORD][10]	:= E_ModbusFunction.WriteSingleRegister;	
// Frequency
arrAddressWrite[iCTRL_FREQUENCY_WORD][0]	:= 100;
arrAddressWrite[iCTRL_FREQUENCY_WORD][1] 	:= 1;
arrAddressWrite[iCTRL_FREQUENCY_WORD][2]	:= LREAL_TO_WORD( FC_ScaleValue(	rangeRawMin := 0,
																				rangeRawMax := 50,
																				RangeScaleMin :=0,
																				RangeScaleMax := 16384,
																				ValueRaw := lrHzControl)
															 );
arrAddressWrite[iCTRL_FREQUENCY_WORD][10]	:= E_ModbusFunction.WriteSingleRegister;												
iNumAddRegionWrite := 2;
END_METHOD

METHOD PROTECTED MS_Aborting
arrAddressWrite[iCTRL_WORD][2] := VFD_CTRL_STOP_FREE;
SUPER^.MS_Aborting();
END_METHOD

METHOD PROTECTED  MS_RunForward
VAR_INPUT
END_VAR
arrAddressWrite[iCTRL_FREQUENCY_WORD][2] :=  LREAL_TO_WORD( FC_ScaleValue(	rangeRawMin := 0,
																			rangeRawMax := 50,
																			RangeScaleMin :=0,
																			RangeScaleMax := 16384,
																			ValueRaw := lrHzControl) );
SUPER^.MS_RunForward();
END_METHOD

METHOD PROTECTED  MS_RunReverse
VAR_INPUT
END_VAR
arrAddressWrite[iCTRL_FREQUENCY_WORD][2] :=  LREAL_TO_WORD( FC_ScaleValue(	rangeRawMin := 0,
																			rangeRawMax := 50,
																			RangeScaleMin :=0,
																			RangeScaleMax := 16384,
																			ValueRaw := lrHzControl) );
super^.MS_RunReverse();
END_METHOD

END_FUNCTION_BLOCK

// ---- POUs/FB_IPRO_ModbusRTU.TcPOU
(* this FB violate Encapsulation of OOP because it still Developing and test to understand how this device work
-------------------------read the document bellow---------------------------------------------------------------*)
FUNCTION_BLOCK FB_IPRO_ModbusRTU EXTENDS FB_ModbusSlave IMPLEMENTS I_Ipro_MotorPower;
VAR_INPUT
END_VAR
VAR_OUTPUT
END_VAR
VAR
	eState : E_IPro_State;
	// bit  read and write modbus 
	bControlModeSwitchCommand	: BOOL;// write p4.15
	bFieldbusEnableServoCommand	:  BOOL;// write p4.11 // anable or disable
	eControlMode				: E_IProCtrlMode;
	lrPositivePositionSoftwareLimit : LREAL;
	lrNagativePositionSoftwareLimit	: LREAL;
	//bClearAbsEncoderMultiturn		: BOOL; should be just config by driver soft
	// dont change value in lrMaxSpeedLimitOfControlModeSwitch
	lrMaxSpeedLimitOfControlModeSwitch	: LREAL := 100;// speed in position mode 	//P0.90// 1180 (*Set the max. running speed during positioning when switching from speed mode or torque mode to position mode under position/speed, position/torque compound mode.*)
	lrPositionCmd					: LREAL;// p4.12 // reference unit // 10000 / rotary
	lrSpeedCmd						: LREAL;// p4.13r/ minute
	lrTorqueCmd						: LREAL; //p4.14 // %
	lrMaxSpeed						: LREAL; // 10x r/ min p4.31 // r/ minute
	lrMaxTorque						: LREAL; // p0.10 % 
	bEmergenCyStop					: BOOL;// 4.23, 1846/ 16 bit //If P4.10 is 1, this parameter can be used to set emergency stop command.
	ePositionCmdModeSelection		: E_IPro_PositionCmdModeSelection;//  not send , it set by ipro soft
	// Read modbus
	lrSpeedFeedback					: LREAL;	// r0.00
	lrTorqueFeedback				: LREAL;	// r0.06
	lrPositionFeedback				: LREAL;// r0.02
	nFaultCode						: INT; // r0.99
	eSystemStatus					: E_IProStatus; // r0.30
	eCurrentMode					: E_IProCurrentMode ;// r0.32 0: Position mode
											// 1: speed mode
											// 2: torque Mode
	ePositionCmdModeSelectionFeedback		: E_IPro_PositionCmdModeSelection;// check if ePositionCmdModeSelection is success write
	// Break ctrol DO
	fbBreakCtrl						: FB_DigitalOutput;									
	(* Generic *)
	//bFirstCycle				: BOOL := TRUE;					(* First cycle bit *)
	sUnit 					: STRING;						(* Measurement units *)
	TempData_Word2real : U_Word2Real;
	TempData_Word2Dint	: U_Word2Dint;
	TempData_Word2Int	: U_Word2Int;

	bInit: BOOL;
	bHome: BOOL;
	bBusy: BOOL;
	bMoveAbsolute: BOOL;
	bReset: BOOL;
	bMoveTorque: BOOL;
	// StopDone
	bStopped: BOOL;
	// StopRequest
	bStop: BOOL;
	lrHomePosition: LREAL;
	// home done
	bHomed: BOOL;
	// Init Done
	bInited: BOOL;
	// MoveAbs Done
	bMoveAbsoluted: BOOL;
	// MoveTorque Done
	bMoveTorqued: BOOL;
	// Abort Request
	bAbort: BOOL;
	bError: BOOL;
	bActive: BOOL;
	bReallyError	: BOOL;// because of bError maybe incorrect because noise information return by Modbus
	tonConfirmReallyError : TON;
	timeConfirmReallyError : TIME := T#15S;
	lrPositivePositionLimit : LREAL;
	lrNagativePositionLimit : LREAL;
END_VAR

(*-------------------Document-------------
	1 set param in drive soft
	2 if set the control mode is different than Curren control mode on the Drive, The drive need restart by drive soft OR turn off power
	3 if the control mode swith command is TRUE, the current control mode will change according to the second mode if eControlMode have
	for example eControlMode = PositionTorque, when bControlModeSwitchCommand = false , currentmode is Position, else current mode is torque if it can
*)

bActive := eState >= IPRO_READY_INITIALIZED;
StateMachine();

bError := nFaultCode <> 0
		OR iModbusErrorID <> MODBUSERROR_NO_ERROR;
CASE eState OF
	IPRO_INITIALIZING..IPRO_RESET_DONE, IPRO_ABORTING:
		tonConfirmReallyError(
			IN := bError,
			PT := timeConfirmReallyError,
			Q => bReallyError 
		);
END_CASE

PROPERTY Active : bool
GET
Active := bActive;
END_GET
END_PROPERTY

{attribute 'monitoring' := 'variable'}
PROPERTY Busy : bool
GET
Busy := bBusy;
END_GET
END_PROPERTY

PROPERTY ControlMode : E_IProCtrlMode
GET
END_GET
SET
IF eState = IPRO_UNINITIALIZED THEN
	THIS^.eControlMode := ControlMode;
END_IF
END_SET
END_PROPERTY

PROPERTY ControlModeSwitchCmd : bool
GET
ControlModeSwitchCmd := bControlModeSwitchCommand;
END_GET
END_PROPERTY

METHOD Convert : BOOL
VAR_INPUT
	iRegionNo	:	INT;
	pReadData	:	POINTER TO word;
END_VAR
VAR
	iLoop		: 	INT;
	TempData	:	 U_Word2Dint;
	TempData_w2i	: U_Word2Int;
	TempData_Int	: INT;
END_VAR
	TempData.iWord[0] := pReadData[0];
	TempData.iWord[1] := pReadData[1];
	TempData_w2i.iWord := pReadData[0];
	TempData_Int := TempData_w2i.iInt;
CASE iRegionNo OF 
	0:// speed 0.1 r/m
		lrSpeedFeedback := DINT_TO_LREAL(TempData.idInt)*0.1;//32 bit
	1:// position unit 1
	
		lrPositionFeedback := DINT_TO_LREAL(TempData.idInt); //64 bit
	2:// torque 0.1
		lrTorqueFeedback := INT_TO_LREAL(TempData_Int)*0.1;
	3:
		eSystemStatus := pReadData[0];
	4:
		eCurrentMode := pReadData[0];
	5:
		nFaultCode := pReadData[0];// must not use word to int

	
END_CASE
END_METHOD

PROPERTY CurrentMode : E_IProCurrentMode
GET
CurrentMode := eCurrentMode;
END_GET
END_PROPERTY

PROPERTY Enable : bool
GET
Enable := bFieldbusEnableServoCommand;
END_GET
END_PROPERTY

PROPERTY Error : bool
GET
Error := bError;
END_GET
END_PROPERTY

PROPERTY ErrorID : REFERENCE TO INT
GET
ErrorID REF= nFaultCode;
END_GET
END_PROPERTY

//Call after Call firstCycleEx
METHOD  FirstCycle // must be call 1 time
VAR_INPUT
	sName : STRING;
	iUnitID : BYTE ; // modbus address of the device : 1- 255
END_VAR
THIS^.sName := sName;
THIS^.iUnitID := iUnitID;

	arrAddressRead[0][0] := 4000;// motor speed FB //0.1 r/min // 4000, 4001
	arrAddressRead[0][1]	:= 2;
	arrAddressRead[0][2] := E_ModbusFunction.ReadHoldingRegisters;
	
	arrAddressRead[1][0] := 4004;// motor position FB// reference unit 
	arrAddressRead[1][1]	:= 4;
	arrAddressRead[1][2] := E_ModbusFunction.ReadHoldingRegisters;
	
	arrAddressRead[2][0] := 4016;// motor Torque FB// reference unit 
	arrAddressRead[2][1]	:= 1;
	arrAddressRead[2][2] := E_ModbusFunction.ReadHoldingRegisters;
	
	arrAddressRead[3][0] := 4064;// System status // 
	arrAddressRead[3][1]	:= 1;
	arrAddressRead[3][2] := E_ModbusFunction.ReadHoldingRegisters;
	
	arrAddressRead[4][0] := 4068;// Current Mode 
	arrAddressRead[4][1]	:= 1;
	arrAddressRead[4][2] := E_ModbusFunction.ReadHoldingRegisters;
	
	arrAddressRead[5][0] := 4198;// FaultCode
	arrAddressRead[5][1]	:= 1;
	arrAddressRead[5][2] := E_ModbusFunction.ReadHoldingRegisters;	
	iNumAddRegionRead := 6;
// write
	arrAddressWrite[0][0] := 1830;// 
	arrAddressWrite[0][1] := 1;
	arrAddressWrite[0][2] := BOOL_TO_WORD(bControlModeSwitchCommand); // disable first
	arrAddressWrite[0][10]	:= E_ModbusFunction.WriteSingleRegister;
	
	arrAddressWrite[1][0] := 1822;// 
	arrAddressWrite[1][1] := 1;
	arrAddressWrite[1][2] :=  BOOL_TO_WORD(bFieldbusEnableServoCommand); // disable first
	arrAddressWrite[1][10]	:= E_ModbusFunction.WriteSingleRegister;
	
	arrAddressWrite[2][0] := 1006;// 
	arrAddressWrite[2][1] := 1;
	arrAddressWrite[2][2] := eControlMode; 
	arrAddressWrite[2][10]	:= E_ModbusFunction.WriteSingleRegister;
	
	arrAddressWrite[3][0] := 1070;//  //32 bit 1070, 1071
	arrAddressWrite[3][1] := 2;
	TempData_Word2Dint.idInt := LREAL_TO_DINT(lrPositivePositionLimit);
	arrAddressWrite[3][2] := TempData_Word2Dint.iWord[0];
	arrAddressWrite[3][3] := TempData_Word2Dint.iWord[1];
	arrAddressWrite[3][10]	:= E_ModbusFunction.WriteMultipleRegisters;
	
	arrAddressWrite[4][0] := 1072;//  //32 bit 1072, 1073
	arrAddressWrite[4][1] := 2;
	TempData_Word2Dint.idInt := LREAL_TO_DINT(lrNagativePositionLimit);
	arrAddressWrite[4][2] := TempData_Word2Dint.iWord[0];
	arrAddressWrite[4][3] := TempData_Word2Dint.iWord[1];
	arrAddressWrite[4][10]	:= E_ModbusFunction.WriteMultipleRegisters;
	
	arrAddressWrite[5][0] := 1180;// 
	arrAddressWrite[5][1] := 1;
	arrAddressWrite[5][2] :=  LREAL_TO_WORD(lrMaxSpeedLimitOfControlModeSwitch); 
	arrAddressWrite[5][10]	:= E_ModbusFunction.WriteSingleRegister;
	
	arrAddressWrite[6][0] := 1824;// 32 bit 1825
	arrAddressWrite[6][1] := 2;
	TempData_Word2Dint.idInt := LREAL_TO_DINT(lrPositionCmd);
	arrAddressWrite[6][2] := TempData_Word2Dint.iWord[0];
	arrAddressWrite[6][3] := TempData_Word2Dint.iWord[1];
	arrAddressWrite[6][10]	:= E_ModbusFunction.WriteMultipleRegisters;
	
	arrAddressWrite[7][0] := 1826;//16 bit
	arrAddressWrite[7][1]	:= 1;
	TempData_Word2Int.iInt := LREAL_TO_INT(lrSpeedCmd);
	arrAddressWrite[7][2] :=  TempData_Word2Int.iWord;
	arrAddressWrite[7][10]	:= E_ModbusFunction.WriteSingleRegister;

	arrAddressWrite[8][0] := 1828;// 16 bit
	arrAddressWrite[8][1]	:= 1;
	TempData_Word2Int.iInt := LREAL_TO_INT(lrTorqueCmd);
	arrAddressWrite[8][2] :=  TempData_Word2Int.iWord;
	arrAddressWrite[8][10]	:= E_ModbusFunction.WriteSingleRegister;
	
	arrAddressWrite[9][0] := 1862;// 1
	arrAddressWrite[9][1]	:= 1;
	TempData_Word2Int.iInt := LREAL_TO_INT(ABS(lrMaxSpeed));
	arrAddressWrite[9][2] :=  TempData_Word2Int.iWord;
	arrAddressWrite[9][10]	:= E_ModbusFunction.WriteSingleRegister;
	
	arrAddressWrite[10][0] := 1020;// 32 bit 1825/ //0.1 PERCENT
	arrAddressWrite[10][1] := 1;
	arrAddressWrite[10][2] :=  LREAL_TO_WORD(ABS(lrMaxTorque));
	arrAddressWrite[10][10]	:= E_ModbusFunction.WriteSingleRegister;
	
	arrAddressWrite[11][0] := 1846;
	arrAddressWrite[11][1] := 1;
	arrAddressWrite[11][2] := BOOL_TO_WORD(THIS^.bEmergenCyStop);
	arrAddressWrite[11][10]	:= E_ModbusFunction.WriteSingleRegister;
	iNumAddRegionWrite := 12;
END_METHOD

METHOD FirstCycleEx : BOOL
VAR_INPUT
	lrPositivePositionLimit : LREAL;
	lrNagativePositionLimit : LREAL;
END_VAR
THIS^.lrPositivePositionLimit := lrPositivePositionLimit;
THIS^.lrNagativePositionLimit := lrNagativePositionLimit;
END_METHOD

{attribute 'monitoring' := 'variable'}
PROPERTY InPosition : bool
GET
InPosition := F_CheckInRange( lrHighLimit := lrPositionFeedback + 20,
						lrLowLimit := lrPositionFeedback - 20,
						lrValue := lrPositionCmd)	;
END_GET
END_PROPERTY

PROPERTY IsHomed : bool
GET
IsHomed := F_CheckInRange( lrHighLimit := lrPositionFeedback + 10,
						lrLowLimit := lrPositionFeedback - 10,
						lrValue := lrHomePosition)	;
END_GET
END_PROPERTY

PROPERTY IsInTorque : bool
GET
isIntorque := F_CheckInRange( lrHighLimit := lrTorqueFeedback + 0.5,// 1%
					lrLowLimit := lrTorqueFeedback -0.5 ,
					lrValue := lrTorqueCmd) ;// +-0.5%	;
END_GET
END_PROPERTY

PROPERTY IsStop : bool // not moving
GET
IsStop := eSystemStatus =  IPRO_STATUS_FAULT;
END_GET
END_PROPERTY

PROPERTY MaxSpeed : lreal// large than 0
GET
MaxSpeed := lrMaxSpeed;
END_GET
SET
IF eState = IPRO_UNINITIALIZED THEN
	lrMaxSpeed := MaxSpeed;
END_IF
END_SET
END_PROPERTY

PROPERTY MaxTorque : Lreal// // % larger than 0
GET
MaxTorque := lrMaxTorque;
END_GET
SET
IF eState = IPRO_UNINITIALIZED THEN
	lrMaxTorque := MaxTorque;
END_IF

arrAddressWrite[10][2] :=  LREAL_TO_WORD(ABS(lrMaxTorque*10));
END_SET
END_PROPERTY

METHOD MR_Abort : BOOL
IF eState >= IPRO_INITIALIZING THEN
	bAbort := TRUE;
	MR_Abort := FALSE;
	eState := IPRO_ABORTING;
ELSIF eState = IPRO_UNINITIALIZED THEN
	bAbort := FALSE;
	MR_Abort := TRUE;
END_IF
END_METHOD

METHOD MR_Home : BOOL // control mode must have Position Mode // actually it the same as MOVE absolute 
VAR_INPUT
	lrHomePosition : LREAL;
END_VAR
IF eState = IPRO_IDLE AND eCurrentMode = IPRO_CURRENT_MODE_POSITION 
AND NOT F_CheckInRange(lrHighLimit := lrHomePosition + 10,
					lrLowLimit := lrHomePosition - 10,
					lrValue := lrPositionFeedback)
THEN 
	bHome := TRUE;
	bHomed := FALSE;
	bBusy := TRUE;
	MR_Home := FALSE;
 	eState := IPRO_HOME;
	THIS^.lrHomePosition := lrHomePosition;
ELSIF  eState = IPRO_IDLE AND eCurrentMode <> IPRO_CURRENT_MODE_POSITION THEN 
	bHome := TRUE;
	bHomed := FALSE;
	bBusy := TRUE;
	MR_Home := FALSE;
 	MS_SwitchMode(eModeChangeTo := IPRO_CURRENT_MODE_POSITION);

ELSIF eState = IPRO_HOME_DONE THEN
	bHomed := TRUE;
	bHome := FALSE;
	bBusy := FALSE;
	MR_Home := TRUE;
END_IF
END_METHOD

(*this must be called 2 times, first: after set All parram in "SetBefor Init" folder and before run FBModbusMaster
							 second : after Modbusmster running and state machine in Init state.*)
METHOD MR_Init : BOOL// need to set control mode carefully, the control mode only work correct if you set p0.03 and restart the driver, and there for if you change control mode cmd during driver power ON, the control mode will not effect


IF eState = IPRO_UNINITIALIZED THEN
	bInit := TRUE;
	bInited := FALSE;
	bBusy := TRUE;
	MR_Init := FALSE;
	eState := IPRO_INITIALIZING;
ELSIF eState = IPRO_READY_INITIALIZED THEN
	bInited := True;
	bInit := FALSE;
	bBusy := FALSE;
	MR_Init := TRUE;
	
END_IF
END_METHOD

METHOD MR_MoveAbsolute : BOOL // control mode must have Position Mode
VAR_INPUT
	lrAbsolutePosition : LREAL;
END_VAR
IF eState = IPRO_IDLE 
AND eCurrentMode = IPRO_CURRENT_MODE_POSITION 
AND NOT F_CheckInRange( lrHighLimit := lrPositionFeedback + 10,
						lrLowLimit := lrPositionFeedback - 10,
						lrValue := lrAbsolutePosition)													
THEN
	lrPositionCmd := lrAbsolutePosition;
	MR_MoveAbsolute := FALSE;
	bBusy := TRUE;
	bMoveAbsolute := TRUE;
	bMoveAbsoluted := FALSE;
	eState := IPRO_MOVE_ABSOLUTE;
ELSIF eState = IPRO_IDLE  AND eCurrentMode <> IPRO_CURRENT_MODE_POSITION THEN
	MR_MoveAbsolute := FALSE;
	bBusy := TRUE;
	bMoveAbsolute := TRUE;
	bMoveAbsoluted := FALSE;
	MS_SwitchMode( eModeChangeTo := IPRO_CURRENT_MODE_POSITION);// if switch mode ok => eCurrentMode = IPRO_CURRENT_MODE_POSITION 

ELSIF eState = IPRO_MOVE_ABSOLUTE_DONE THEN
	bBusy := FALSE;
	bMoveAbsolute := FALSE;
	MR_MoveAbsolute := TRUE;
	bMoveAbsoluted := TRUE;
	
ELSIF  eState = IPRO_IDLE 
	AND eCurrentMode = IPRO_CURRENT_MODE_POSITION 
	AND F_CheckInRange( lrHighLimit := lrPositionFeedback + 10,
							lrLowLimit := lrPositionFeedback - 10,
							lrValue := lrAbsolutePosition)													
	THEN
		bBusy := FALSE;
		bMoveAbsolute := FALSE;
		MR_MoveAbsolute := TRUE;
		bMoveAbsoluted := TRUE;
END_IF
END_METHOD

METHOD MR_MoveTorque : BOOL // control mode must have torque Mode edit :Torque can be change every time if needed;
VAR_INPUT
	lrTorque	: LREAL;// must smaller than max torque
END_VAR

IF eState = IPRO_IDLE
AND eCurrentMode = IPRO_CURRENT_MODE_TORQUE 
AND NOT F_CheckInRange( lrHighLimit := lrTorqueFeedback + 0.5,// 1%
					lrLowLimit := lrTorqueFeedback -0.5 ,
					lrValue := lrTorque) // +-0.5%	
THEN
	bMoveTorque	:= TRUE;
	bMoveTorqued	:= FALSE;
	bBusy := TRUE;
	MR_MoveTorque := FALSE;
	eState := IPRO_MOVE_TORQUE;
	lrTorqueCmd := lrTorque;
ELSIF eState = IPRO_IDLE AND eCurrentMode <>  IPRO_CURRENT_MODE_TORQUE THEN
	MR_MoveTorque := FALSE;
	bBusy := TRUE;
	bMoveTorque := TRUE;
	bMoveTorqued	:= FALSE;
	MS_SwitchMode( eModeChangeTo := IPRO_CURRENT_MODE_TORQUE);// if switch mode ok => eCurrentMode = IPRO_CURRENT_MODE_POSITION 

ELSIF eState = IPRO_IDLE OR eState = IPRO_MOVE_TORQUE_DONE THEN
	bBusy := FALSE;
	bMoveTorque := FALSE;
	MR_MoveTorque := TRUE;
	bMoveTorqued	:= TRUE;
END_IF
END_METHOD

METHOD MR_Reset : BOOL// can't not use this method because i didn't find way to reset
(*IF eState <> IPRO_RESET AND eState <> IPRO_RESET_DONE THEN
	bReset := TRUE;
	MR_Reset := FALSE;
	eState := IPRO_RESET;
ELSIF eState = IPRO_RESET_DONE THEN
	bReset := FALSE;
	MR_Reset := TRUE;
	
END_IF*)
END_METHOD

METHOD MR_Stop : BOOL // carefully because it lead to IPRO_STATUS_FAULT // need to be init again
IF eState >= IPRO_IDLE AND eState <> IPRO_STOP_DONE THEN
	bStop := TRUE;
	bStopped := FALSE;
	MR_Stop := FALSE;
	eState := IPRO_STOP;
	bBusy := TRUE;
ELSIF eState = IPRO_STOP_DONE THEN
	bStop := FALSE;
	bStopped := TRUE;
	MR_Stop := TRUE;
	bBusy := FALSE;
END_IF
END_METHOD

METHOD PROTECTED MS_Aborting// still remain all the params set before init
VAR_INPUT
END_VAR
bFieldbusEnableServoCommand := FALSE;
bEmergenCyStop := false;
arrAddressWrite[1][2] :=  BOOL_TO_WORD(bFieldbusEnableServoCommand);
IF THIS^.eSystemStatus <> IPRO_STATUS_RUN THEN
	eState := IPRO_UNINITIALIZED;
END_IF
END_METHOD

METHOD PROTECTED MS_Home
VAR_INPUT
END_VAR
TempData_Word2Dint.idInt := LREAL_TO_DINT(lrHomePosition);
arrAddressWrite[6][2] := TempData_Word2Dint.iWord[0];
arrAddressWrite[6][3] := TempData_Word2Dint.iWord[1];

IF F_CheckInRange(lrHighLimit := lrHomePosition + 10,
					lrLowLimit := lrHomePosition - 10,
					lrValue := lrPositionFeedback)
THEN
	eState := IPRO_HOME_DONE;
END_IF
END_METHOD

METHOD PROTECTED  MS_HomeDone
VAR_INPUT
END_VAR
IF NOT bHome THEN
	eState := IPRO_IDLE;
END_IF
END_METHOD

METHOD PROTECTED MS_Idle
VAR_INPUT
END_VAR
;
END_METHOD

METHOD PROTECTED MS_Initializing
VAR_INPUT
END_VAR
arrAddressWrite[2][2] := eControlMode; 

TempData_Word2Int.iInt := LREAL_TO_INT(ABS(lrMaxSpeed));
arrAddressWrite[9][2] :=  TempData_Word2Int.iWord;

arrAddressWrite[5][2] :=  LREAL_TO_WORD(lrMaxSpeedLimitOfControlModeSwitch); // unit 1

arrAddressWrite[10][2] :=  LREAL_TO_WORD(ABS(lrMaxTorque*10));

TempData_Word2Dint.idInt := LREAL_TO_DINT(lrNagativePositionSoftwareLimit);
arrAddressWrite[4][2] := TempData_Word2Dint.iWord[0];
arrAddressWrite[4][3] := TempData_Word2Dint.iWord[1];

TempData_Word2Dint.idInt := LREAL_TO_DINT(lrPositivePositionSoftwareLimit);
arrAddressWrite[3][2] := TempData_Word2Dint.iWord[0];
arrAddressWrite[3][3] := TempData_Word2Dint.iWord[1];


// this servo can't reset error by modbus
IF THIS^.eSystemStatus = IPRO_STATUS_READY THEN // Ignor the faultcode AND nFaultCode = 0  THEN
	bFieldbusEnableServoCommand := TRUE;
	arrAddressWrite[1][2] :=  BOOL_TO_WORD(bFieldbusEnableServoCommand);
END_IF
 
IF eSystemStatus = IPRO_STATUS_RUN THEN
	eState := IPRO_READY_INITIALIZED;
END_IF
END_METHOD

METHOD PROTECTED MS_MoveAbsolute
VAR_INPUT
END_VAR
TempData_Word2Dint.idInt := LREAL_TO_DINT(lrPositionCmd);
arrAddressWrite[6][2] := TempData_Word2Dint.iWord[0];
arrAddressWrite[6][3] := TempData_Word2Dint.iWord[1];

IF F_CheckInRange(lrHighLimit := lrPositionCmd + 10,
					lrLowLimit := lrPositionCmd - 10,
					lrValue := lrPositionFeedback)
THEN
	eState := IPRO_MOVE_ABSOLUTE_DONE;
END_IF
END_METHOD

METHOD PROTECTED MS_MoveAbsoluteDone
VAR_INPUT
END_VAR
IF NOT bMoveAbsolute THEN
	eState := IPRO_IDLE;
END_IF
END_METHOD

METHOD PROTECTED MS_MoveTorque
VAR_INPUT
END_VAR
TempData_Word2Int.iInt := LREAL_TO_INT(lrTorqueCmd *10);
arrAddressWrite[8][2] :=  TempData_Word2Int.iWord;
(* should by pass this one if not, it can't receive new Torque
IF F_CheckInRange( lrHighLimit := lrTorqueFeedback + 0.5,// 1%
					lrLowLimit := lrTorqueFeedback -0.5 ,
					lrValue := lrTorqueCmd) 
THEN
	eState := IPRO_MOVE_TORQUE_DONE;
END_IF*)
eState := IPRO_MOVE_TORQUE_DONE;
END_METHOD

METHOD PROTECTED MS_MoveTorqueDone
VAR_INPUT
END_VAR
IF NOT bMoveTorque THEN
	eState := IPRO_IDLE;
END_IF
END_METHOD

METHOD PROTECTED MS_ReadyInitialized
VAR_INPUT
END_VAR
IF NOT bInit THEN
	eState := IPRO_IDLE;
END_IF
END_METHOD

METHOD PROTECTED MS_Reset
VAR_INPUT
END_VAR
END_METHOD

METHOD PROTECTED MS_ResetDone
VAR_INPUT
END_VAR
END_METHOD

METHOD PROTECTED MS_Stop
VAR_INPUT
END_VAR
bEmergenCyStop := TRUE;
arrAddressWrite[11][2] := BOOL_TO_WORD(THIS^.bEmergenCyStop);
IF eSystemStatus = IPRO_STATUS_FAULT THEN
	eState := IPRO_STOP_DONE;
END_IF
END_METHOD

METHOD PROTECTED MS_StopDone
VAR_INPUT
END_VAR
IF NOT bStop THEN
	eState := IPRO_UNINITIALIZED;
END_IF
END_METHOD

METHOD PROTECTED MS_SwitchMode : BOOL;
VAR_INPUT
	eModeChangeTo	: E_IProCurrentMode; // False is the first mode , TRUE is Seconde Mode in Control mode
END_VAR


CASE THIS^.eControlMode OF
	
	IPRO_CTRL_MODE_POSITION_TORQUE:
		IF eModeChangeTo = IPRO_CURRENT_MODE_POSITION THEN
			bControlModeSwitchCommand := FALSE;
		ELSIF eModeChangeTo = IPRO_CURRENT_MODE_TORQUE THEN
			bControlModeSwitchCommand := TRUE;
		END_IF
	IPRO_CTRL_MODE_POSITION_SPEED:
		IF eModeChangeTo = IPRO_CURRENT_MODE_POSITION THEN
			bControlModeSwitchCommand := FALSE;
		ELSIF eModeChangeTo = IPRO_CURRENT_MODE_SPEED THEN
			bControlModeSwitchCommand := TRUE;
		END_IF
	IPRO_CTRL_MODE_SPEED_TORQUE:
		IF eModeChangeTo = IPRO_CURRENT_MODE_SPEED THEN
			bControlModeSwitchCommand := FALSE;
		ELSIF eModeChangeTo = IPRO_CURRENT_MODE_TORQUE THEN
			bControlModeSwitchCommand := TRUE;
		END_IF
	
END_CASE

arrAddressWrite[0][2] :=  BOOL_TO_WORD(bControlModeSwitchCommand); 

IF eCurrentMode = eModeChangeTo THEN
	MS_SwitchMode := TRUE;
ELSE
	MS_SwitchMode := FALSE;	
END_IF
END_METHOD

METHOD PROTECTED MS_Uninitalized
VAR_INPUT
END_VAR
END_METHOD

PROPERTY NagativePositionLimit : lreal
GET
NagativePositionLimit := lrNagativePositionSoftwareLimit;
END_GET
SET
IF eState = IPRO_UNINITIALIZED THEN
	lrNagativePositionSoftwareLimit := NagativePositionLimit;
END_IF
END_SET
END_PROPERTY

PROPERTY PositionCmd : lreal
GET
PositionCmd := lrPositionCmd;
END_GET
END_PROPERTY

PROPERTY PositionFeedBack : lreal
GET
PositionFeedBack := lrPositionFeedback;
END_GET
END_PROPERTY

PROPERTY PositionModeSelectionCmd : E_IPro_PositionCmdModeSelection
GET
PositionModeSelectionCmd := ePositionCmdModeSelection;
END_GET
END_PROPERTY

PROPERTY PositionModeSelectionFeedback : E_IPro_PositionCmdModeSelection
GET
PositionModeSelectionFeedback := ePositionCmdModeSelectionFeedback;
END_GET
END_PROPERTY

PROPERTY PositionPositiveLimit : lreal
GET
PositionPositiveLimit := lrPositivePositionSoftwareLimit;
END_GET
SET
IF eState = IPRO_UNINITIALIZED THEN
	lrPositivePositionSoftwareLimit := PositionPositiveLimit;
END_IF
END_SET
END_PROPERTY

PROPERTY ReallyError : bool
SET
ReallyError := bReallyError;
END_SET
END_PROPERTY

PROPERTY SpeedCmd : LREAL // r/ minute
GET
SpeedCmd := lrSpeedCmd;
END_GET
SET
lrSpeedCmd := SpeedCmd;
TempData_Word2Int.iInt := LREAL_TO_INT(lrSpeedCmd*10);
arrAddressWrite[7][2] :=  TempData_Word2Int.iWord;
END_SET
END_PROPERTY

PROPERTY SpeedFeedback : Lreal
GET
SpeedFeedback := lrSpeedFeedback;
END_GET
END_PROPERTY

PROPERTY State : E_IPro_State
GET
State := eState;
END_GET
END_PROPERTY

METHOD PROTECTED StateMachine
VAR_INPUT
END_VAR

VAR

END_VAR
CASE eState OF
		IPRO_UNINITIALIZED:
		MS_Uninitalized();
		
	IPRO_INITIALIZING:
		MS_Initializing();
		
	IPRO_READY_INITIALIZED:
		MS_ReadyInitialized();
		
	IPRO_IDLE:
		MS_Idle();
		
	IPRO_HOME:
		MS_Home();
		
	IPRO_HOME_DONE:
		MS_HomeDone();
		
	IPRO_MOVE_ABSOLUTE:
		MS_MoveAbsolute();
	
	IPRO_MOVE_ABSOLUTE_DONE:
		MS_MoveAbsoluteDone();
		
	IPRO_MOVE_TORQUE:
		MS_MoveTorque();
		
	IPRO_MOVE_TORQUE_DONE: 
		MS_MoveTorqueDone();
	
	IPRO_STOP:
		MS_Stop();
	
	IPRO_STOP_DONE:
		MS_StopDone();
		
	IPRO_RESET:
		MS_Reset();
	
	IPRO_RESET_DONE:
		MS_ResetDone();
		
	IPRO_ABORTING:
		MS_Aborting();
	

		
END_CASE
END_METHOD

PROPERTY Status : E_IProStatus
GET
Status := eSystemStatus;
END_GET
END_PROPERTY

PROPERTY TorqueCmd : lreal // %
GET
TorqueCmd :=  lrTorqueCmd ;
END_GET
END_PROPERTY

PROPERTY TorqueFeedback : lreal
GET
TorqueFeedback := lrTorqueFeedback;
END_GET
END_PROPERTY

END_FUNCTION_BLOCK
